TYPE CyclicVel_CMD_typ :
STRUCT
	
	Start 		: BOOL;
	Disable 	: BOOL;
	
END_STRUCT
END_TYPE

(* stored: Version 1.1.0.1, ProductVersion 3.1.4024.3
   DUT CyclicVel_CMD_typ: Id {9d21f657-929c-013f-1d86-1ec4783ad18b} *)
